// TIA Portal V20 export
DATA_BLOCK "DB_VisuColor"   // DB2
// stored: Access Published, MemoryReserve 100, Namespace Global
   VAR
      Line : Struct
         A1 : Struct
            Conveyor : Array[_.gMinA1.._.gMaxA1] of Int;
         END_STRUCT;
         B1 : Struct
            Conveyor : Array[_.gMinB1.._.gMaxB1] of Int;
         END_STRUCT;
         C1 : Struct
            Conveyor : Array[_.gMinC1.._.gMaxC1] of Int;
         END_STRUCT;
         D1 : Struct
            Conveyor : Array[_.gMinD1.._.gMaxD1] of Int;
         END_STRUCT;
      END_STRUCT;
   END_VAR
BEGIN
END_DATA_BLOCK
